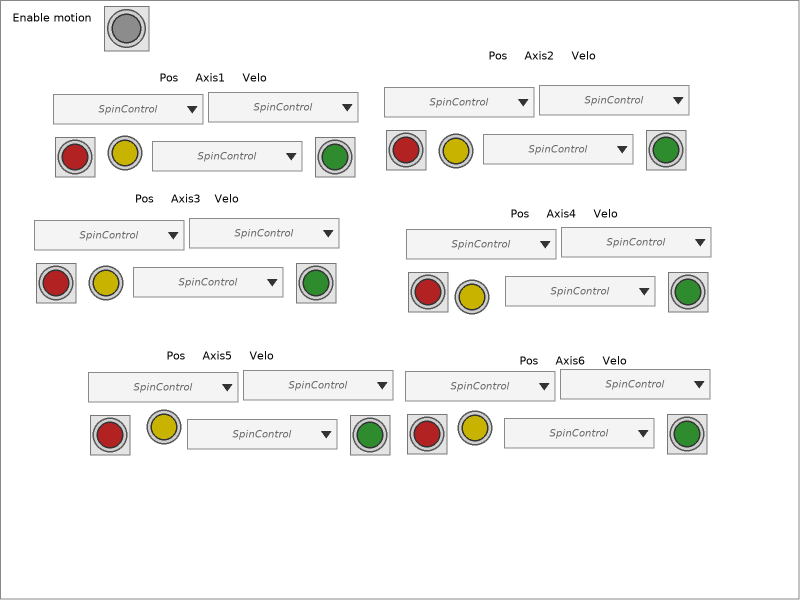
VISUALIZATION StandMotors  // 800x600
    PushSwitch (104,2 45x53), variable: MAIN.bEnable, behaviour: TOGGLE, style: Switch-PushSwitch-Gray
    Lamp1 (105,133 40x40), variable: GVL_ver.AXIS1_Brake_q_disabled, style: Lamp-Lamp1-Yellow
    Label (8,3 88x30), "Enable motion"
    Lamp1 (436,131 40x40), variable: GVL_ver.AXIS2_Brake_q_disabled, style: Lamp-Lamp1-Yellow
    Lamp1 (86,263 40x40), variable: GVL_ver.AXIS3_Brake_q_disabled, style: Lamp-Lamp1-Yellow
    Lamp1 (452,277 40x40), variable: GVL_ver.AXIS4_Brake_q_disabled, style: Lamp-Lamp1-Yellow
    Lamp1 (144,407 40x40), variable: GVL_ver.AXIS5_Brake_q_disabled, style: Lamp-Lamp1-Yellow
    Lamp1 (455,408 40x40), variable: GVL_ver.AXIS6_Brake_q_disabled, style: Lamp-Lamp1-Yellow
    SpinControl (406,229 150x30), variable: Axis4.rPosition
    PushSwitch (408,272 40x40), variable: Axis4.boHalt, behaviour: TOGGLE, style: Switch-PushSwitch-Red
    PushSwitch (668,272 40x40), variable: Axis4.boMoveAbsolute, behaviour: TOGGLE, style: Switch-PushSwitch-Green
    SpinControl (505,276 150x30), variable: Axis4.roPosition
        p1653691745: 0.05
    SpinControl (561,227 150x30), variable: Axis4.rVelocity
        p1653691745: 0.05
    Label (489,199 150x30), "Pos Axis4 Velo"
    Label (498,346 150x30), "Pos Axis6 Velo"
    Label (145,341 150x30), "Pos Axis5 Velo"
    PushSwitch (36,263 40x40), variable: Axis3.boHalt, behaviour: TOGGLE, style: Switch-PushSwitch-Red
    SpinControl (34,220 150x30), variable: Axis3.rPosition
    PushSwitch (296,263 40x40), variable: Axis3.boMoveAbsolute, behaviour: TOGGLE, style: Switch-PushSwitch-Green
    SpinControl (133,267 150x30), variable: Axis3.roPosition
        p1653691745: 0.05
    SpinControl (189,218 150x30), variable: Axis3.rVelocity
        p1653691745: 0.05
    PushSwitch (386,130 40x40), variable: Axis2.boHalt, behaviour: TOGGLE, style: Switch-PushSwitch-Red
    SpinControl (384,87 150x30), variable: Axis2.rPosition
    PushSwitch (646,130 40x40), variable: Axis2.boMoveAbsolute, behaviour: TOGGLE, style: Switch-PushSwitch-Green
    SpinControl (483,134 150x30), variable: Axis2.roPosition
        p1653691745: 0.05
    SpinControl (539,85 150x30), variable: Axis2.rVelocity
        p1653691745: 0.05
    PushSwitch (55,137 40x40), variable: Axis1.boHalt, behaviour: TOGGLE, style: Switch-PushSwitch-Red
    SpinControl (53,94 150x30), variable: Axis1.rPosition
    PushSwitch (315,137 40x40), variable: Axis1.boMoveAbsolute, behaviour: TOGGLE, style: Switch-PushSwitch-Green
    SpinControl (152,141 150x30), variable: Axis1.roPosition
        p1653691745: 0.05
    SpinControl (208,92 150x30), variable: Axis1.rVelocity
        p1653691745: 0.05
    PushSwitch (407,414 40x40), variable: Axis6.boHalt, behaviour: TOGGLE, style: Switch-PushSwitch-Red
    SpinControl (405,371 150x30), variable: Axis6.rPosition
    PushSwitch (667,414 40x40), variable: Axis6.boMoveAbsolute, behaviour: TOGGLE, style: Switch-PushSwitch-Green
    SpinControl (504,418 150x30), variable: Axis6.roPosition
        p1653691745: 0.05
    SpinControl (560,369 150x30), variable: Axis6.rVelocity
        p1653691745: 0.05
    PushSwitch (90,415 40x40), variable: Axis5.boHalt, behaviour: TOGGLE, style: Switch-PushSwitch-Red
    SpinControl (88,372 150x30), variable: Axis5.rPosition
    PushSwitch (350,415 40x40), variable: Axis5.boMoveAbsolute, behaviour: TOGGLE, style: Switch-PushSwitch-Green
    SpinControl (187,419 150x30), variable: Axis5.roPosition
        p1653691745: 0.05
    SpinControl (243,370 150x30), variable: Axis5.rVelocity
        p1653691745: 0.05
    Label (112,184 150x30), "Pos Axis3 Velo"
    Label (467,41 150x30), "Pos Axis2 Velo"
    Label (138,63 150x30), "Pos Axis1 Velo"
END_VISUALIZATION

(* stored: Version 1.1.0.1, ProductVersion 3.1.4022.3
   Visu StandMotors: Id {2362f43e-7307-4c02-abc0-6879981ddffb} *)
